SUBAPPLICATION Uebung_006a2 (* 2x SR und T-Flip-Flop mit IE *)
  (* Standard: 61499-2; Description: Copyright (c) 2023 Meisterschulen am Ostbahnhof This program and the accompanying materials are made available under the terms of the Eclipse Public License 2.0 which is available at https://www.eclipse.org/legal/epl-2.0/ SPDX-License-Identifier: EPL-2.0 *)
  (* Version 1.0, 2023-10-23, Franz Höpfinger, Meisterschulen am Ostbahnhof *)
  IMPORT logiBUS::io::DI::logiBUS_DI;
  IMPORT logiBUS::io::DQ::logiBUS_DO;
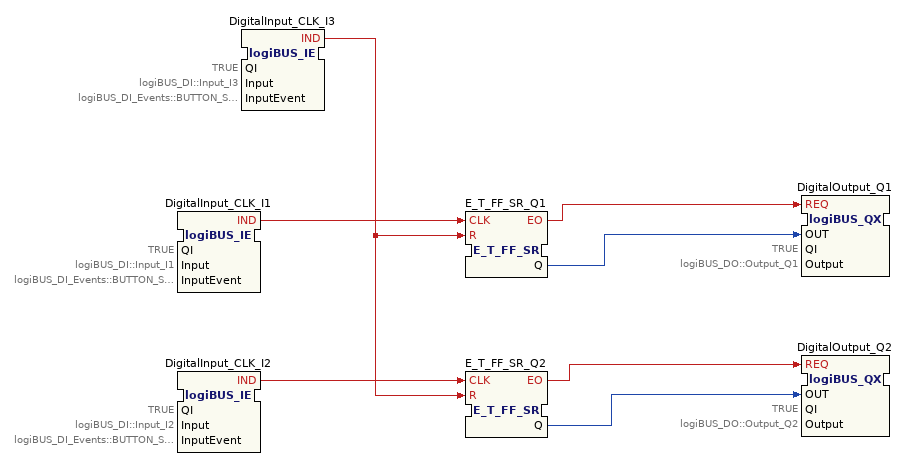
  FBS
    DigitalOutput_Q1 : logiBUS::io::DQ::logiBUS_QX(QI := TRUE, Output := logiBUS_DO::Output_Q1);
    DigitalInput_CLK_I1 : logiBUS_IE(QI := TRUE, Input := logiBUS_DI::Input_I1, InputEvent := logiBUS_DI_Events::BUTTON_SINGLE_CLICK);
    DigitalInput_CLK_I2 : logiBUS_IE(QI := TRUE, Input := logiBUS_DI::Input_I2, InputEvent := logiBUS_DI_Events::BUTTON_SINGLE_CLICK);
    E_T_FF_SR_Q1 : iec61499::events::E_T_FF_SR;
    DigitalInput_CLK_I3 : logiBUS_IE(QI := TRUE, Input := logiBUS_DI::Input_I3, InputEvent := logiBUS_DI_Events::BUTTON_SINGLE_CLICK);
    E_T_FF_SR_Q2 : iec61499::events::E_T_FF_SR;
    DigitalOutput_Q2 : logiBUS::io::DQ::logiBUS_QX(QI := TRUE, Output := logiBUS_DO::Output_Q2);
  END_FBS
  EVENT_CONNECTIONS
    E_T_FF_SR_Q1.EO TO DigitalOutput_Q1.REQ;
    E_T_FF_SR_Q2.EO TO DigitalOutput_Q2.REQ;
    DigitalInput_CLK_I1.IND TO E_T_FF_SR_Q1.CLK;
    DigitalInput_CLK_I2.IND TO E_T_FF_SR_Q2.CLK;
    DigitalInput_CLK_I3.IND TO E_T_FF_SR_Q2.R;
    DigitalInput_CLK_I3.IND TO E_T_FF_SR_Q1.R;
  END_CONNECTIONS
  DATA_CONNECTIONS
    E_T_FF_SR_Q1.Q TO DigitalOutput_Q1.OUT;
    E_T_FF_SR_Q2.Q TO DigitalOutput_Q2.OUT;
  END_CONNECTIONS
END_SUBAPPLICATION
